{attribute 'linkalways'}
{attribute 'no_explicit_call' := 'do not call this POU directly'}
FUNCTION_BLOCK GlobalNamespace
VAR_STAT // singleton
	lastInstanceNamespace : STRING;
END_VAR

METHOD FB_init : BOOL
VAR_INPUT
	bInitRetains : BOOL; // if TRUE, the retain variables are initialized (warm start / cold start)
	bInCopyCode : BOOL;  // if TRUE, the instance afterwards gets moved into the copy code (online change)
	Instance : I_Instance;
END_VAR
IF Instance.NameSpace = '' THEN
	RETURN;
END_IF

lastInstanceNamespace := Instance.NameSpace;
END_METHOD

METHOD PUBLIC GetLastInstanceNamespace : String
VAR_INPUT
END_VAR
GetLastInstanceNamespace := lastInstanceNamespace;
END_METHOD

END_FUNCTION_BLOCK

(* stored: Version 1.1.0.1, ProductVersion 3.1.4024.11
   POU GlobalNamespace: Id {bb55475b-70c8-4652-b733-872ee003630c}, SpecialFunc None
   Folder Constructor: Id {ee7b2540-8d7d-4343-9aa1-e49b03a0768e}
   Method FB_init: Id {c985942f-5c5d-4663-8ed1-43d0a8e98009}
   Method GetLastInstanceNamespace: Id {06108602-e9ec-4bf1-ab0d-8b430815b4ba} *)
